FUNCTION_BLOCK E_CTD (* Event-Driven Down Counter *)
  (* Standard: 61499-1-A.x; Classification: Event-driven blocks; Function: Down-counter; Description: Copyright (c) 2017 fortiss GmbH This program and the accompanying materials are made available under the terms of the Eclipse Public License 2.0 which is available at https://www.eclipse.org/legal/epl-2.0/ SPDX-License-Identifier: EPL-2.0 *)
  (* Version 1.0, 2017-09-22, Alois Zoitl, fortiss GmbH, initial API and implementation and/or initial documentation *)
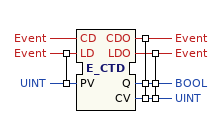
  EVENT_INPUT
    CD; (* Count Down *)
    LD WITH PV; (* Load counter value *)
  END_EVENT
  EVENT_OUTPUT
    CDO WITH Q, CV; (* Count Down Output Event *)
    LDO WITH Q, CV; (* Reset Output Event *)
  END_EVENT
  VAR_INPUT
    PV : UINT; (* Preset Value *)
  END_VAR
  VAR_OUTPUT
    Q : BOOL; (* CV <= 0 *)
    CV : UINT;
  END_VAR
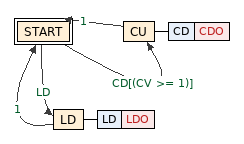
  EC_STATES
    START;
    CU : CD -> CDO;
    LD : LD -> LDO;
  END_STATES
  EC_TRANSITIONS
    START TO CU := CD[(CV >= 1)];
    CU TO START := 1;
    START TO LD := LD;
    LD TO START := 1;
  END_TRANSITIONS
  ALGORITHM CD IN ST: (* Count Down *)
CV := CV - 1;
Q := (CV <= 0);
  END_ALGORITHM
  ALGORITHM LD IN ST: (* Load *)
CV := PV;
Q:= (CV <= 0);
  END_ALGORITHM
END_FUNCTION_BLOCK
